FUNCTION_BLOCK FB_Wheel
VAR_INPUT
END_VAR
VAR_OUTPUT
END_VAR
VAR
END_VAR

PROPERTY Speed : real
GET
END_GET
SET
END_SET
END_PROPERTY

END_FUNCTION_BLOCK

(* stored: Version 1.1.0.1, ProductVersion 3.1.4024.11
   POU FB_Wheel: Id {2106bd09-116e-4a48-a995-6720f2929ced}, SpecialFunc None
   Property Speed: Id {e24d56b3-8c6b-4fd8-aa63-ec2620b3e6c9}
   Get Get: Id {e6c5b242-37c8-43bd-b7a8-7de7b41891a7}
   Set Set: Id {bb985251-504e-43cb-b6ee-00514bda0071} *)
